FUNCTION F_VNx_EnsureGray : HRESULT
VAR_INPUT
	ipSrcImage		:	ITcVnImage;
	ipDestImage		:	REFERENCE TO ITcVnImage;
	hrPrev			:	HRESULT;
END_VAR
VAR
	hr				:	HRESULT;
	stFormat		:	TcVnPixelFormat;	
END_VAR

// Check params
IF FAILED(hrPrev) THEN
	F_VNx_EnsureGray := hrPrev;
	RETURN;
END_IF

IF ipSrcImage = 0 THEN
	F_VNx_EnsureGray := Tc2_System.E_HRESULTAdsErr.INVALIDPARM;
	RETURN;
END_IF

// Processing
hr := F_VN_GetPixelFormat(ipSrcImage, stFormat, hr);

CASE stFormat.nChannels OF
1:
	// To get 2 independent images a copy is necessary in this case
	hr := F_VN_CopyImage(ipSrcImage, ipDestImage, hr);
3:
	hr := F_VN_ConvertColorSpace(ipSrcImage, ipDestImage, TCVN_CST_RGB_TO_GRAY, hr);
4:
	hr := F_VN_ConvertColorSpace(ipSrcImage, ipDestImage, TCVN_CST_RGBA_TO_GRAY, hr);
ELSE
	hr := Tc2_System.E_HRESULTAdsErr.INCOMPATIBLE;
END_CASE

// Return
F_VNx_EnsureGray := hr;
RETURN;

END_FUNCTION

(* stored: Version 1.1.0.1, ProductVersion 3.1.4024.6
   POU F_VNx_EnsureGray: Id {f7bc7c63-ceb2-4499-bbd6-e2f9b9ba07f0}, SpecialFunc None *)
